PROGRAM MAIN
VAR
	iCount : UINT;
	fbSlaveStateChange : FB_EcSetSlaveState;
	AmsNetId : AMSNETID;
	Ams : T_AmsNetId;
	bTrigger : BOOL;
	State : WORD;
	test123 AT %Q* : USINT;
	vonKlemme AT %I* : USINT;
	
	CurrentState : ST_EcSlaveState;
END_VAR

iCount := GVL.iTest;
Ams := '10.183.66.136.4.1';
test123 := TO_USINT(iCount); 
fbSlaveStateChange(
	 sNetId := Ams,
	 nSlaveAddr := 1001,
	 bExecute := bTrigger,
	 tTimeout := T#10S,
	 reqState := State,
	 
	 bBusy =>,
	 bError =>,
	 nErrId =>,
	 currState=>
	 );
	 
CurrentState := fbSlaveStateChange.currState;

IF CurrentState.deviceState = State AND bTrigger THEN
	bTrigger := FALSE;
END_IF

END_PROGRAM

(* stored: Version 1.1.0.1, ProductVersion 3.1.4024.12
   POU MAIN: Id {c474b279-45ae-49a1-aa1e-ee0327b7f910}, SpecialFunc None *)
